FUNCTION_BLOCK PUBLIC FB_ADD
VAR_INPUT
END_VAR
VAR_OUTPUT
END_VAR
VAR
END_VAR

END_FUNCTION_BLOCK

(* stored: Version 1.1.0.1, ProductVersion 3.1.4024.12
   POU FB_ADD: Id {b5d921c4-ce65-4c4e-86a8-3f0b4223d0dc}, SpecialFunc None *)
